# EPICS substitutions: bkhApp/Db/bkhMotrSaveRestore.substitutions
#==============================================================================
file "bkhMotrSaveRestore.template"
{pattern{N,  M, PREC}
        {15, 1,    3}
        {15, 2,    3}
        {15, 3,    3}
        {15, 4,    3}
        {15, 5,    3}
        {15, 6,    3}
}
